FUNCTION_BLOCK FB67
TITLE = 'fault_Z4'
AUTHOR : CB

VAR
	fault_Z4CONV1VAD : FB66;
END_VAR


BEGIN


NETWORK
TITLE =
//
//	fault/fault_Z4/fault_Z4CONV1VAD
CALL #fault_Z4CONV1VAD;




END_FUNCTION_BLOCK
